(*

short summary
=============
a candy vending machine for the picky eaters. 
It tries to provide candies that match the desired candy type. 

legal notes
===========
SPDX-FileCopyrightText: © 2024 ekvip automation GmbH <info@ekvip.de>
SPDX-License-Identifier: Apache-2.0
For details check: Apache-2.0_

.. _Apache-2.0: https://www.apache.org/licenses/LICENSE-2.0

*)

FUNCTION_BLOCK FINAL PickyCandyMachine EXTENDS AbstractCandyMachine

(*

short summary
=============
want some, get some
this method provides the candies

legal notes
===========
SPDX-FileCopyrightText: © 2024 ekvip automation GmbH <info@ekvip.de>
SPDX-License-Identifier: Apache-2.0
For details check: Apache-2.0_

.. _Apache-2.0: https://www.apache.org/licenses/LICENSE-2.0

*)

METHOD  getNewCandy :REFERENCE TO AbstractCandy
VAR_INPUT
	(*preferred candy type, it must be a pure candy type *)
	candyType	:CandyTypes;
END_VAR
VAR
	(* the __NEW operator requires a stricktly typed pointer *)
	alpenliebe			:POINTER TO Alpenliebe;		
	(* the __NEW operator requires a stricktly typed pointer *)
	altoids				:POINTER TO Altoids;
	(* the __NEW operator requires a stricktly typed pointer *)
	bobsStripes			:POINTER TO BobsSweetStripes;
	(* the __NEW operator requires a stricktly typed pointer *)
	candyCorn			:POINTER TO BrachsCandyCorn;
	(* the __NEW operator requires a stricktly typed pointer *)
	chupChups			:POINTER TO ChupaChups;
	(* the __NEW operator requires a stricktly typed pointer *)
	goldbears			:POINTER TO Goldbears;
	(* the __NEW operator requires a stricktly typed pointer *)
	mAndMs				:POINTER TO MnMs;	
	(* the __NEW operator requires a stricktly typed pointer *)
	skittles			:POINTER TO SkittlesSour;
	(* the __NEW operator requires a stricktly typed pointer *)
	poppins				:POINTER TO Poppins;
	(* the __NEW operator requires a stricktly typed pointer *)
	snickers			:POINTER TO SnickersBar;
	(* the __NEW operator requires a stricktly typed pointer *)
	twizzlers			:POINTER TO TwizzlersLicorizeTwists;
	(* the __NEW operator requires a stricktly typed pointer *)
	gobstopper			:POINTER TO WonkaGobstopper;
	(* return value is just a candy *)
	candy				:POINTER TO AbstractCandy;
END_VAR
getNewCandy REF= 0;
RETURN(THIS^.isCandyTypeInvalidForMachine(candyType));

CASE candyType OF
CandyTypes.CANDY_BARS:
	snickers := __NEW(SnickersBar());
	candy := snickers;
CandyTypes.CANDY_CORN:
	candyCorn := __NEW(BrachsCandyCorn());
	candy := candyCorn;
CandyTypes.CANDY_STICKS:
	bobsStripes := __NEW(BobsSweetStripes());
	candy := bobsStripes;
CandyTypes.CARAMEL_CANDY:
	alpenliebe := __NEW(Alpenliebe());
	candy := alpenliebe;
CandyTypes.CHOCOLATE_CANDY:
	mAndMs := __NEW(MnMs());
	candy := mAndMs;
CandyTypes.GUMMY_CANDY:;		
	goldbears := __NEW(Goldbears());
	candy := goldbears;		
CandyTypes.HARD_CANDY:
	poppins := __NEW(Poppins());
	candy := poppins;		
CandyTypes.LOLLIPOPS:
	chupChups := __NEW(ChupaChups());
	candy := chupChups;
CandyTypes.JAWBREAKERS:
	gobstopper := __NEW(WonkaGobstopper());
	candy := gobstopper;
CandyTypes.LICORICE_CANDY:
	twizzlers := __NEW(TwizzlersLicorizeTwists());
	candy := twizzlers;
CandyTypes.MINTS:
	altoids := __NEW(Altoids());
	candy := altoids;
CandyTypes.SOUR_CANDY:
	skittles := __NEW(SkittlesSour());
	candy := skittles;
ELSE
	RETURN;	
END_CASE

RETURN(candy <= 0);
getNewCandy REF= candy^;
END_METHOD

END_FUNCTION_BLOCK

(* stored: Version 1.1.0.1
   POU PickyCandyMachine: Id {d95ab528-6c9f-4339-a849-b428ebd2aa58}, SpecialFunc None
   Method getNewCandy: Id {85fa8b75-7e34-4d56-822c-fe33a97f5db0} *)
